// Mitsubishi GX Works2 project: 0630tlfflsej dmddydehdwkr 1   PLC: Q02/Q02H

PROGRAM MAIN
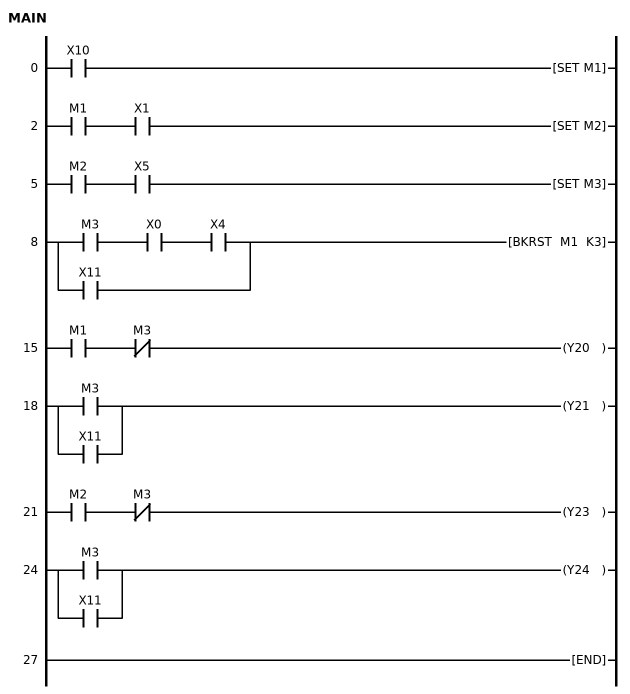
0     LD      X10
      SET     M1
2     LD      M1
      AND     X1
      SET     M2
5     LD      M2
      AND     X5
      SET     M3
8     LD      M3
      AND     X0
      AND     X4
      OR      X11
      BKRST   M1 K3
15    LD      M1
      ANI     M3
      OUT     Y20
18    LD      M3
      OR      X11
      OUT     Y21
21    LD      M2
      ANI     M3
      OUT     Y23
24    LD      M3
      OR      X11
      OUT     Y24
27    END
END_PROGRAM

PROGRAM MAIN1
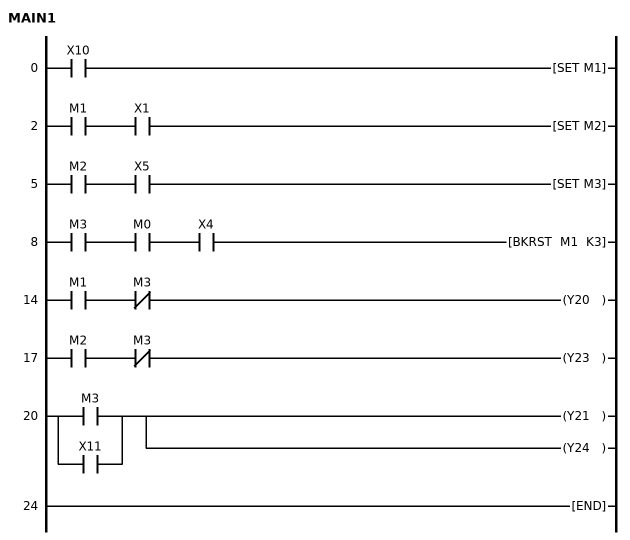
0     LD      X10
      SET     M1
2     LD      M1
      AND     X1
      SET     M2
5     LD      M2
      AND     X5
      SET     M3
8     LD      M3
      AND     M0
      AND     X4
      BKRST   M1 K3
14    LD      M1
      ANI     M3
      OUT     Y20
17    LD      M2
      ANI     M3
      OUT     Y23
20    LD      M3
      OR      X11
      OUT     Y21
      OUT     Y24
24    END
END_PROGRAM
